// SIMATIC STEP 7 (V5.x) project HW8 - PLC - Problem 3
// CPU: CPU 314C-2 DP
// station: Hardware
// station: SIMATIC 300(1)
// station: P_ADR_BUS
// program: S7 Program(1)

SYMBOL_TABLE
"Mode_OFF"	I 0.0	BOOL
"Mode_Manual"	I 0.1	BOOL
"Mode_Auto"	I 0.2	BOOL
"PB_S1_Extend"	I 0.3	BOOL
"PB_S2_Retract"	I 0.4	BOOL
"LS_Retracted"	I 0.5	BOOL
"LS_Extended"	I 0.6	BOOL
"State_OFF"	M 0.0	BOOL
"State_Manual"	M 0.1	BOOL
"State_Auto"	M 0.2	BOOL
"Valve_Extend"	Q 0.0	BOOL
"Valve_Retract"	Q 0.1	BOOL
END_SYMBOL_TABLE

ORGANIZATION_BLOCK OB 1
TITLE = "Main Program Sweep (Cycle)"
//HW8 - PLC - Problem 3
VERSION : 0.1
VAR_TEMP
  OB1_EV_CLASS : BYTE ;	//Bits 0-3 = 1 (Coming event), Bits 4-7 = 1 (Event class 1)
  OB1_SCAN_1 : BYTE ;	//1 (Cold restart scan 1 of OB 1), 3 (Scan 2-n of OB 1)
  OB1_PRIORITY : BYTE ;	//Priority of OB Execution
  OB1_OB_NUMBR : BYTE ;	//1 (Organization block 1, OB1)
  OB1_RESERVED_1 : BYTE ;	//Reserved for system
  OB1_RESERVED_2 : BYTE ;	//Reserved for system
  OB1_PREV_CYCLE : INT ;	//Cycle time of previous OB1 scan (milliseconds)
  OB1_MIN_CYCLE : INT ;	//Minimum cycle time of OB1 (milliseconds)
  OB1_MAX_CYCLE : INT ;	//Maximum cycle time of OB1 (milliseconds)
  OB1_DATE_TIME : DATE_AND_TIME ;	//Date and time OB1 started
END_VAR
BEGIN
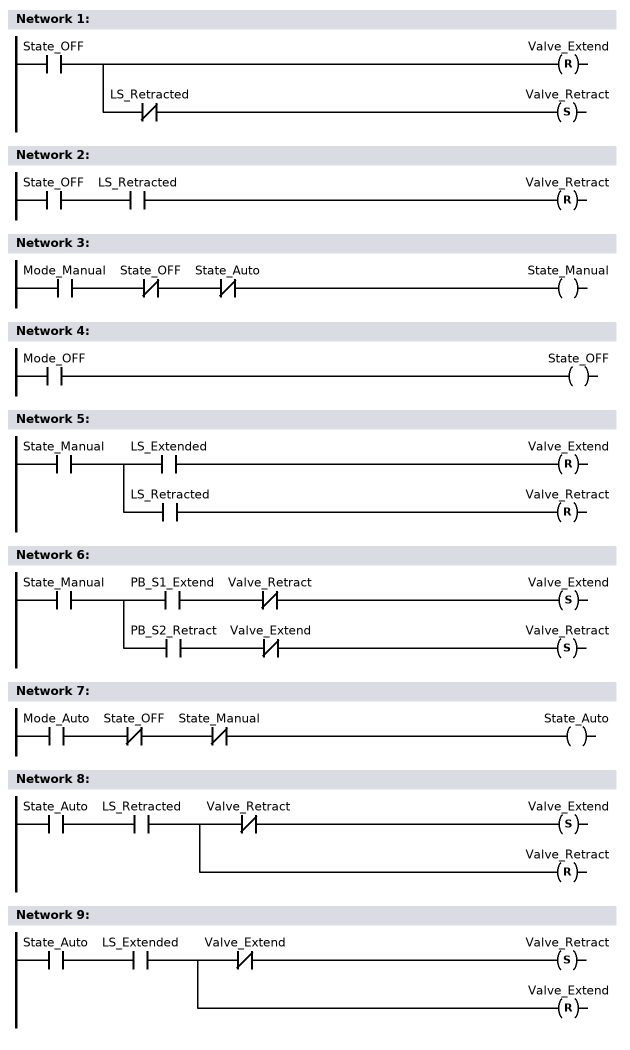
NETWORK
TITLE =
      A     "State_OFF";
      =     L 20.0;
      A     L 20.0;
      BLD   102;
      R     "Valve_Extend";
      A     L 20.0;
      AN    "LS_Retracted";
      S     "Valve_Retract";
NETWORK
TITLE =
      A     "State_OFF";
      A     "LS_Retracted";
      R     "Valve_Retract";
NETWORK
TITLE =
      A     "Mode_Manual";
      AN    "State_OFF";
      AN    "State_Auto";
      =     "State_Manual";
NETWORK
TITLE =
      A     "Mode_OFF";
      =     "State_OFF";
NETWORK
TITLE =
      A     "State_Manual";
      =     L 20.0;
      A     L 20.0;
      A     "LS_Extended";
      R     "Valve_Extend";
      A     L 20.0;
      A     "LS_Retracted";
      R     "Valve_Retract";
NETWORK
TITLE =
      A     "State_Manual";
      =     L 20.0;
      A     L 20.0;
      A     "PB_S1_Extend";
      AN    "Valve_Retract";
      S     "Valve_Extend";
      A     L 20.0;
      A     "PB_S2_Retract";
      AN    "Valve_Extend";
      S     "Valve_Retract";
NETWORK
TITLE =
      A     "Mode_Auto";
      AN    "State_OFF";
      AN    "State_Manual";
      =     "State_Auto";
NETWORK
TITLE =
      A     "State_Auto";
      A     "LS_Retracted";
      =     L 20.0;
      A     L 20.0;
      AN    "Valve_Retract";
      S     "Valve_Extend";
      A     L 20.0;
      BLD   102;
      R     "Valve_Retract";
NETWORK
TITLE =
      A     "State_Auto";
      A     "LS_Extended";
      =     L 20.0;
      A     L 20.0;
      AN    "Valve_Extend";
      S     "Valve_Retract";
      A     L 20.0;
      BLD   102;
      R     "Valve_Extend";
END_ORGANIZATION_BLOCK
